FUNCTION_BLOCK FB_DivertFullMonitor

VAR_IN_OUT
	Divert 			: ST_Divert;
END_VAR

VAR
	LastFullTime	: REAL;
	nFullTime : UINT;
	Cfg_FullTime: TIME := T#2S;
END_VAR

// Calculate and set the merge clear timer
IF LastFullTime <> Divert.Config.FullTime THEN
	LastFullTime := Divert.Config.FullTime;
	nFullTime := REAL_TO_UINT(LastFullTime * 1000); 
	Cfg_FullTime := UINT_TO_TIME(nFullTime);
END_IF

// Set the Full time, according to the Full-Time
Divert.FullTimer(PT := Cfg_FullTime);

// Test for Full
Divert.FullTimer(IN := Divert.FullPE);

IF Divert.FullTimer.Q THEN
	Divert.Full := TRUE;
ELSE
	Divert.Full := FALSE;
END_IF

END_FUNCTION_BLOCK

(* stored: Version 1.1.0.1, ProductVersion 3.1.4024.4
   POU FB_DivertFullMonitor: Id {61f277c4-19da-4b53-b17c-0567be4f20bc}, SpecialFunc None *)
